// TwinCAT 3 PLC project PLC
// ProgramVersion: 3.1.4026.19
// libraries:
//   Tc2_MC2, * (Beckhoff Automation GmbH)
//   Tc2_Standard, * (Beckhoff Automation GmbH)
//   Tc2_System, * (Beckhoff Automation GmbH)
// project tree:
//   GVLs/ GVL_Safety.TcGVL
//   / PlcTask.TcTTO
//   POUs/ MAIN.TcPOU
// real-time tasks:
//   TASK PlcTask: cycle T#10ms, priority 20, ADS port 350
// variable links:
//   PLC/PLC Instance <-> PLC/PLC Instance
//     PlcTask Inputs/GVL_Safety.bSafety_MotorPowerOK <-> PlcTask Outputs/GVL_Safety.bSafety_EStopPressed

CONFIGURATION PLC
    RESOURCE PLC ON TwinCAT3
        TASK PlcTask(INTERVAL := T#10ms, PRIORITY := 20);
        PROGRAM MAIN WITH PlcTask : MAIN;
    END_RESOURCE
END_CONFIGURATION

// ---- GVLs/GVL_Safety.TcGVL
{attribute 'qualified_only'}
VAR_GLOBAL
	bSafety_EStopPressed AT %Q* : BOOL;
	bSafety_ResetCmd AT %Q* : BOOL;
	bSafety_MotorPowerOK AT %I* : BOOL;
END_VAR

// ---- POUs/MAIN.TcPOU
PROGRAM MAIN
VAR
    axisVirtualMotor : AXIS_REF;
    fbPower          : MC_Power;
    bEnable          : BOOL;
END_VAR

IF NOT GVL_Safety.bSafety_EStopPressed THEN
    GVL_Safety.bSafety_MotorPowerOK := FALSE; 
    
ELSIF GVL_Safety.bSafety_ResetCmd THEN
    GVL_Safety.bSafety_MotorPowerOK := TRUE;
END_IF


fbPower(
    Axis := axisVirtualMotor,

    Enable := bEnable AND GVL_Safety.bSafety_MotorPowerOK, 
    Enable_Positive := bEnable AND GVL_Safety.bSafety_MotorPowerOK,
    Enable_Negative := bEnable AND GVL_Safety.bSafety_MotorPowerOK,
    Override := 100.0
);

END_PROGRAM
